(* IEC 61131-3 sources: IRIS-Project/LASAL CONTROL SOFTWARE/LasalProject_2025_09_12/Runtime/%LASALAPPDATA%/Runtime/Library/Loader/Class/MMServer, 1 file *)

(* ---- MMServer.st ---- *)
(*!
<Class
	Name               = "MMServer"
	Revision           = "0.0"
	RealtimeTask       = "false"
	CyclicTask         = "false"
	BackgroundTask     = "false"
	Sigmatek           = "true"
	OSInterface        = "false"
	HighPriority       = "false"
	Automatic          = "false"
	UpdateMode         = "Prescan"
	SharedCommandTable = "true"
	Objectsize         = "(690,120)">
	<Channels>
	</Channels>
	<RevDoku>
		<Owner Company="Sigmatek" Author="FimLuc"/>
		<Dokumentation Revision="0.0" Date="2015-10-07" Author="FimLuc" Company="Sigmatek" Description="erstellt"/>
	</RevDoku>
	<Network Name="MMServer">
		<!-- List of Components in this network -->
		<Components>
			<Object
				Name       = "_base"
				Class      = "MMServerImpl"
				Position   = "(698,120)"
				Visualized = "false">
				<Channels>
					<Server Name="Data"/>
					<Client Name="DataBuffer"/>
					<Client Name="DataBufferOut"/>
				</Channels>
			</Object>
		</Components>
		<Comments>
		</Comments>
		<!-- List of Connections in this network -->
		<Connections>
			<Connection Source="this.Data" Destination="_base.Data" Vertices="(1696,210),(1524,210),"/>
		</Connections>
		<!-- Headerfiles -->
		<Options>
		</Options>
	</Network>
</Class>
*)
#pragma using MMServerImpl

MMServer : CLASS
: MMServerImpl
  //Servers:
  //Clients:
  //Variables:
  //Functions:
  //Tables:
	FUNCTION @STD
		VAR_OUTPUT
			ret_code	: CONFSTATES;
		END_VAR;
	FUNCTION GLOBAL TAB @CT_;
END_CLASS;
